// TIA Portal V19 export
FUNCTION_BLOCK "CallGlobal"   // FB48, LAD
TITLE = CallGlobal
// All blocks that provide data to the DB Global.Data are called here. That includes blocks to generate system data as well as blocks that connect handle multiple HMIs.
// stored: IsIECCheckEnabled true, MemoryReserve 100, SetENOAutomatically true
   VAR
      statClockSysMemOld { ExternalWritable := 'False'} : Byte;   // Old value system memory evaluation / Alter Wert Systeminformationsspeicher auswertung
      instLAF_PowerOnOff { ExternalWritable := 'False'} : "LAF_PowerOnOff";
      instLAF_ClockGen { ExternalWritable := 'False'} : "LAF_ClockGenerator";
      instLSNTP_Server { ExternalWritable := 'False'} : "LSNTP_Server";
      instLAF_SpecialFunctionsManager { S7_SetPoint := 'True'} : "LAF_SpecialFunctionsManager";
   END_VAR
   VAR_TEMP
      tempResultXor : Byte;   // Interim result of XOR operation / Zwischenergebnis von XOR Anweisung
      tempPosPulse : Byte;   // Interim result puls calculation / Zwischenergebnis von Pulsauswertung
   END_VAR
   VAR CONSTANT
      RESET_BUTTON__COULD_BE_ADDED_HERE : Bool := false;   // Placeholder for a potential global reset button
   END_VAR
BEGIN

REGION Network 1: Global Acknowledge
   // The global acknowledge command from the hmi button is assigned to Global.Data.general.acknowledge: This bit it forwarded to all underlaying modules
   // If a hard-wired global reset button exists, it can
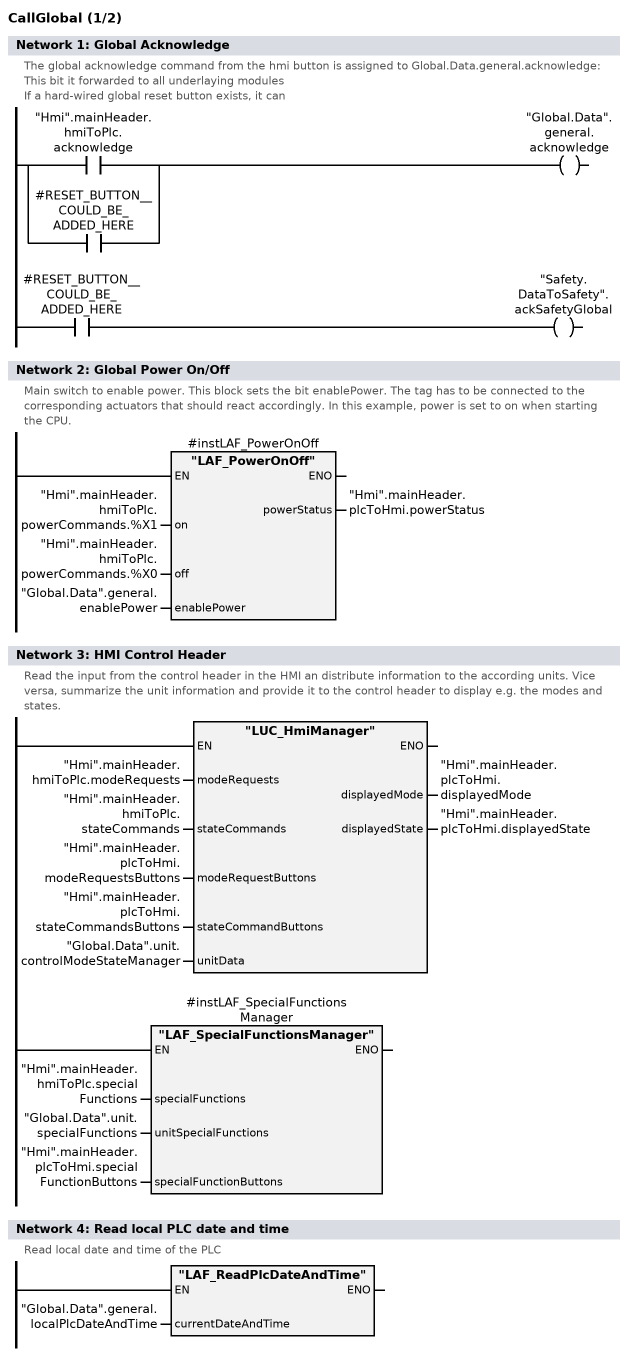
   RUNG wire#powerrail
      Contact( "Hmi".mainHeader.hmiToPlc.acknowledge )
      wire#w1
      Coil( "Global.Data".general.acknowledge )
   END_RUNG
   RUNG wire#powerrail
      Contact( #RESET_BUTTON__COULD_BE_ADDED_HERE )
   END_RUNG wire#w1
   RUNG wire#powerrail
      Contact( #RESET_BUTTON__COULD_BE_ADDED_HERE )
      Coil( "Safety.DataToSafety".ackSafetyGlobal )
   END_RUNG
   // the same network as SCL:
   "Global.Data".general.acknowledge := "Hmi".mainHeader.hmiToPlc.acknowledge OR #RESET_BUTTON__COULD_BE_ADDED_HERE;
   "Safety.DataToSafety".ackSafetyGlobal := #RESET_BUTTON__COULD_BE_ADDED_HERE;
END_REGION

REGION Network 2: Global Power On/Off
   // Main switch to enable power. This block sets the bit enablePower. The tag has to be connected to the corresponding actuators that should react accordingly. In this example, power is set to on when starting the CPU.
   RUNG wire#powerrail
      #instLAF_PowerOnOff(on := "Hmi".mainHeader.hmiToPlc.powerCommands.%X1, off := "Hmi".mainHeader.hmiToPlc.powerCommands.%X0, enablePower := "Global.Data".general.enablePower, powerStatus => "Hmi".mainHeader.plcToHmi.powerStatus)
   END_RUNG
   // the same network as SCL:
   #instLAF_PowerOnOff(on := "Hmi".mainHeader.hmiToPlc.powerCommands.%X1,   // "LAF_PowerOnOff"
                       off := "Hmi".mainHeader.hmiToPlc.powerCommands.%X0,
                       enablePower := "Global.Data".general.enablePower,
                       powerStatus => "Hmi".mainHeader.plcToHmi.powerStatus);
END_REGION

REGION Network 3: HMI Control Header
   // Read the input from the control header in the HMI an distribute information to the according units. Vice versa, summarize the unit information and provide it to the control header to display e.g. the modes and states.
   RUNG wire#powerrail
      "LUC_HmiManager"(modeRequests := "Hmi".mainHeader.hmiToPlc.modeRequests, stateCommands := "Hmi".mainHeader.hmiToPlc.stateCommands, modeRequestButtons := "Hmi".mainHeader.plcToHmi.modeRequestsButtons, stateCommandButtons := "Hmi".mainHeader.plcToHmi.stateCommandsButtons, unitData := "Global.Data".unit.controlModeStateManager, displayedMode => "Hmi".mainHeader.plcToHmi.displayedMode, displayedState => "Hmi".mainHeader.plcToHmi.displayedState)
   END_RUNG
   RUNG wire#powerrail
      #instLAF_SpecialFunctionsManager(specialFunctions := "Hmi".mainHeader.hmiToPlc.specialFunctions, unitSpecialFunctions := "Global.Data".unit.specialFunctions, specialFunctionButtons := "Hmi".mainHeader.plcToHmi.specialFunctionButtons)
   END_RUNG
   // the same network as SCL:
   "LUC_HmiManager"(modeRequests := "Hmi".mainHeader.hmiToPlc.modeRequests,
                    stateCommands := "Hmi".mainHeader.hmiToPlc.stateCommands,
                    modeRequestButtons := "Hmi".mainHeader.plcToHmi.modeRequestsButtons,
                    stateCommandButtons := "Hmi".mainHeader.plcToHmi.stateCommandsButtons,
                    unitData := "Global.Data".unit.controlModeStateManager,
                    displayedMode => "Hmi".mainHeader.plcToHmi.displayedMode,
                    displayedState => "Hmi".mainHeader.plcToHmi.displayedState);
   #instLAF_SpecialFunctionsManager(specialFunctions := "Hmi".mainHeader.hmiToPlc.specialFunctions,   // "LAF_SpecialFunctionsManager"
                           unitSpecialFunctions := "Global.Data".unit.specialFunctions,
                           specialFunctionButtons := "Hmi".mainHeader.plcToHmi.specialFunctionButtons);
END_REGION

REGION Network 4: Read local PLC date and time
   // Read local date and time of the PLC
   RUNG wire#powerrail
      "LAF_ReadPlcDateAndTime"(currentDateAndTime := "Global.Data".general.localPlcDateAndTime)
   END_RUNG
   // the same network as SCL:
   "LAF_ReadPlcDateAndTime"(currentDateAndTime := "Global.Data".general.localPlcDateAndTime);
END_REGION

REGION Network 5: Create clock bits / Takt Bits erstellen
   // The clock bits are generated instead of the HW clock memory byte of the PLC. Due to the use of software units, the ussage of system and clock memory bytes isn't possible. / Die Taktbits werden erzeugt anstelle der HW Taktmerker Byte der SPS. Durch die verwendung von Softwareunits ist der Zugriff auf die System und Taktmerker nicht möglich.
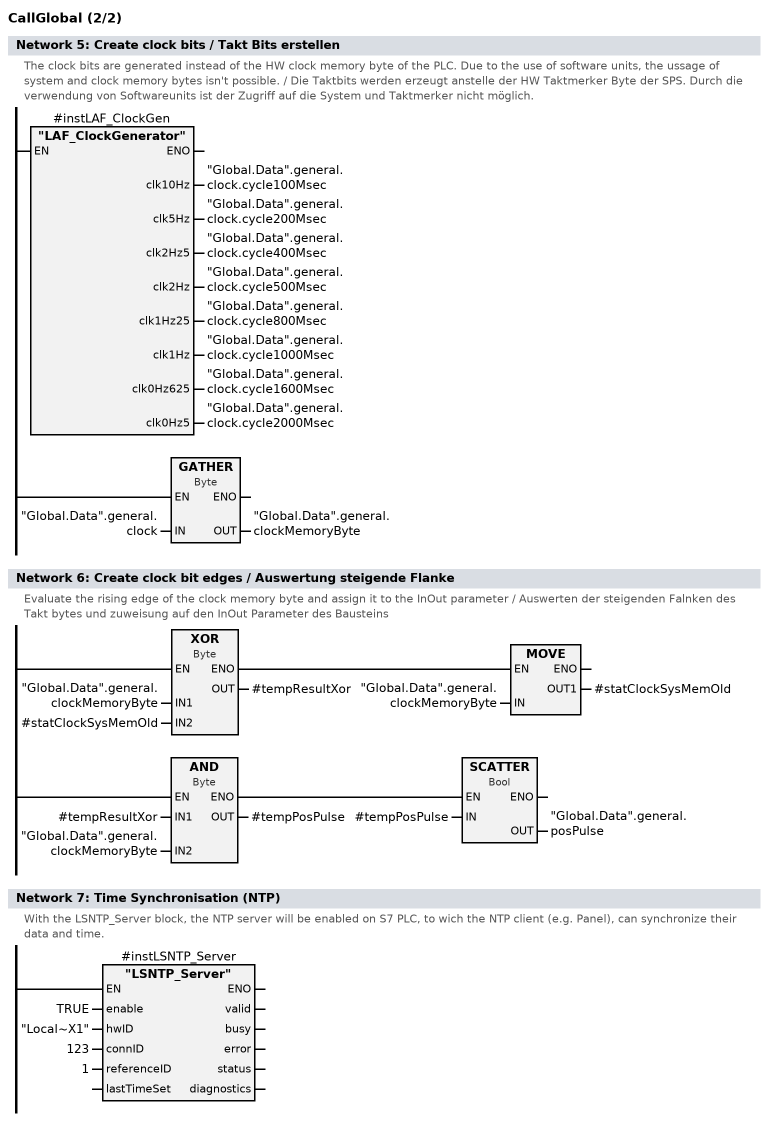
   RUNG wire#powerrail
      #instLAF_ClockGen(clk10Hz => "Global.Data".general.clock.cycle100Msec, clk5Hz => "Global.Data".general.clock.cycle200Msec, clk2Hz5 => "Global.Data".general.clock.cycle400Msec, clk2Hz => "Global.Data".general.clock.cycle500Msec, clk1Hz25 => "Global.Data".general.clock.cycle800Msec, clk1Hz => "Global.Data".general.clock.cycle1000Msec, clk0Hz625 => "Global.Data".general.clock.cycle1600Msec, clk0Hz5 => "Global.Data".general.clock.cycle2000Msec)
   END_RUNG
   RUNG wire#powerrail
      { S7_Templates := "[dest_type := Byte, src_type := Bool]" } GATHER(IN := "Global.Data".general.clock, OUT => "Global.Data".general.clockMemoryByte)
   END_RUNG
   // the same network as SCL:
   #instLAF_ClockGen(clk10Hz => "Global.Data".general.clock.cycle100Msec,   // "LAF_ClockGenerator"
                     clk5Hz => "Global.Data".general.clock.cycle200Msec,
                     clk2Hz5 => "Global.Data".general.clock.cycle400Msec,
                     clk2Hz => "Global.Data".general.clock.cycle500Msec,
                     clk1Hz25 => "Global.Data".general.clock.cycle800Msec,
                     clk1Hz => "Global.Data".general.clock.cycle1000Msec,
                     clk0Hz625 => "Global.Data".general.clock.cycle1600Msec,
                     clk0Hz5 => "Global.Data".general.clock.cycle2000Msec);
   GATHER(IN := "Global.Data".general.clock, OUT => "Global.Data".general.clockMemoryByte);
END_REGION

REGION Network 6: Create clock bit edges / Auswertung steigende Flanke
   // Evaluate the rising edge of the clock memory byte and assign it to the InOut parameter / Auswerten der steigenden Falnken des Takt bytes und zuweisung auf den InOut Parameter des Bausteins
   #tempResultXor := "Global.Data".general.clockMemoryByte XOR #statClockSysMemOld;
   #statClockSysMemOld := "Global.Data".general.clockMemoryByte;
   #tempPosPulse := #tempResultXor AND "Global.Data".general.clockMemoryByte;
   SCATTER(IN := #tempPosPulse, OUT => "Global.Data".general.posPulse);
END_REGION

REGION Network 7: Time Synchronisation (NTP)
   // With the LSNTP_Server block, the NTP server will be enabled on S7 PLC, to wich the NTP client (e.g. Panel), can synchronize their data and time.
   RUNG wire#powerrail
      #instLSNTP_Server(enable := TRUE, hwID := "Local~X1", connID := 123, referenceID := 1, lastTimeSet :=, valid =>, busy =>, error =>, status =>, diagnostics =>)
   END_RUNG
   // the same network as SCL:
   #instLSNTP_Server(enable := TRUE, hwID := "Local~X1", connID := 123, referenceID := 1);   // "LSNTP_Server"
END_REGION
END_FUNCTION_BLOCK
